FUNCTION_BLOCK F_SPLIT_LTOD (* split LTIME_OF_DAY *)
  (* Standard: 61131-3; Classification: standard character and string function; Description: Copyright (c) 2013 TU Wien ACIN and others. This program and the accompanying materials are made available under the terms of the Eclipse Public License 2.0 which is available at https://www.eclipse.org/legal/epl-2.0/ SPDX-License-Identifier: EPL-2.0 Some portions generated by Gemini CLI *)
  (* Version 1.0, 2026-01-31, Franz Höpfinger, HR Agrartechnik GmbH, initial API and implementation and/or initial documentation *)
  PACKAGE iec61131::charString;
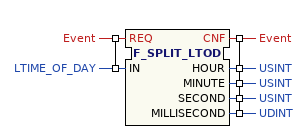
  EVENT_INPUT
    REQ WITH IN; (* Service Request *)
  END_EVENT
  EVENT_OUTPUT
    CNF WITH HOUR, MINUTE, SECOND, MILLISECOND; (* Confirmation of Requested Service *)
  END_EVENT
  VAR_INPUT
    IN : LTIME_OF_DAY; (* Input LTIME_OF_DAY *)
  END_VAR
  VAR_OUTPUT
    HOUR : USINT; (* Hour *)
    MINUTE : USINT; (* Minute *)
    SECOND : USINT; (* Second *)
    MILLISECOND : UDINT; (* Millisecond *)
  END_VAR
  EC_STATES
    REQ : REQ -> CNF;
  END_STATES
  ALGORITHM REQ IN ST:
SPLIT_LTOD(IN, HOUR, MINUTE, SECOND, MILLISECOND);
  END_ALGORITHM
END_FUNCTION_BLOCK
